{attribute 'GeneratedUsingTerminal: AT2050-0501-0017'}
{attribute addProperty BoxType "AT2050-0501-0017"}
{attribute addProperty Id "A_0088_AT2050_5501_0017_AT2050_5501AT2050_33A3DF1B80"}
{attribute addProperty CRC "2706044123"}
{attribute addProperty Size "80"}
TYPE A_0056_AT2050_0501_0017_A14AF4DB EXTENDS AT2050_A7FEA1CF :
STRUCT
	{attribute addProperty Name "A_0088_AT2050_5501_0017_AT2050_5501"}
	{attribute addProperty PreviousPort "A_0056(AT2050-0501-0017) : B"}
	A_0088_AT2050_5501_0017_AT2050_5501 : AT2050_33A3DF1B;
END_STRUCT
END_TYPE

(* stored: Version 1.2.0.0, ProductVersion 3.1.4024.9
   DUT A_0056_AT2050_0501_0017_A14AF4DB: Id {a9c38681-b37a-4cec-be39-c83552e61394} *)
